TYPE ST_System_FBT_Stellwert :
STRUCT
	Anford_Pumpe		: BOOL;
	Anford_Regelventil	: BOOL;
	Temp_Vorl			: REAL;
END_STRUCT
END_TYPE

(* stored: Version 1.1.0.1, ProductVersion 3.1.4024.9
   DUT ST_System_FBT_Stellwert: Id {b9af9dd3-4136-4630-9387-cc897b412bf7} *)
